TYPE "AppControl"
VERSION : 0.1
   STRUCT
      start : Bool;
      stop : Bool;
   END_STRUCT;

END_TYPE

